{attribute 'GeneratedUsingTerminal: BK1250-0000-0000'}
{attribute addProperty BoxType "BK1250-0000-0000"}
{attribute addProperty Id "Term_397_KL1002KL1002_BB38DA8F0"}
{attribute addProperty CRC "165800773"}
{attribute addProperty Size "0"}
TYPE A_0014_BK1250_0000_0000_09E1EB45 EXTENDS BK1250_A2FCADE7 :
STRUCT
	{attribute addProperty Name "Term_397_KL1002"}
	Term_397_KL1002 : KL1002_BB38DA8F;
END_STRUCT
END_TYPE

(* stored: Version 1.2.0.0, ProductVersion 3.1.4024.9
   DUT A_0014_BK1250_0000_0000_09E1EB45: Id {d826cbf6-5ec9-454c-8722-11d1522b423b} *)
